// TwinCAT 3 PLC project PLC_Modbus_TCP
// ProgramVersion: 3.1.4024.0
// libraries:
//   Tc2_ModbusSrv, * (Beckhoff Automation GmbH)
//   Tc2_Standard, * (Beckhoff Automation GmbH)
//   Tc2_System, * (Beckhoff Automation GmbH)
//   Tc3_Module, * (Beckhoff Automation GmbH)
// project tree:
//   / PlcTask.TcTTO
//   POUs/ FB_Counter.TcPOU, FB_ReadCoilsExample.TcPOU, FB_WriteRegsExample.TcPOU, MAIN.TcPOU
// real-time tasks:
//   TASK PlcTask: cycle T#10ms, priority 20, ADS port 350

CONFIGURATION PLC_Modbus_TCP
    RESOURCE PLC ON TwinCAT3
        TASK PlcTask(INTERVAL := T#10ms, PRIORITY := 20);
        PROGRAM MAIN WITH PlcTask : MAIN;
    END_RESOURCE
END_CONFIGURATION

// ---- POUs/MAIN.TcPOU
PROGRAM MAIN
VAR
	fbWriteRegs : FB_WriteRegsExample;
	fbWriteRwgs_2 : FB_WriteRegsExample; 
END_VAR

fbWriteRegs();
fbWriteRwgs_2();

END_PROGRAM

// ---- POUs/FB_WriteRegsExample.TcPOU
FUNCTION_BLOCK FB_WriteRegsExample
VAR
	fbWriteRegisters : FB_MBWriteRegs;
	nWriteValueArray : ARRAY[0..9] OF INT;
	wWriteRegsValueConvertToWord : WORD;
	eWriteState : (WAIT, TRIGGER, WRITE);
	fbTriggerStart : R_TRIG;
	fbTriggerStop : R_TRIG;
	//cbLength: UINT;
	
END_VAR

fbTriggerStart();
IF fbTriggerStart.Q THEN
	IF eWriteState = WAIT THEN
		 eWriteState := TRIGGER;
	END_IF
END_IF
IF fbTriggerStop.CLK THEN
	fbWriteRegisters(bExecute := FALSE);
	eWriteState := WAIT;
END_IF
CASE eWriteState OF
	WAIT : 
	// NOTHING
	TRIGGER : 
	 //wWriteRegsValueConvertToWord := TO_WORD(nWriteValueInt);
	 (*fbWriteRegisters(
		sIPAddr:= '192.168.10.1', 
		nTCPPort:= 502, 
		nUnitID:= 16#FF, 
		nMBAddr:= 0, 
		nValue:= wWriteRegsValueConvertToWord, 
		bExecute:= TRUE, 
		tTimeout:= , 
		bBusy=> , 
		bError=> , 
		nErrId=> ); *)
	fbWriteRegisters(
		sIPAddr:= '192.168.10.1', 
		nTCPPort:= 502, 
		nUnitID:= 16#FF, 
		nQuantity:= 10, 
		nMBAddr:= 0, 
		cbLength:= SIZEOF(nWriteValueArray), 
		pSrcAddr:= ADR(nWriteValueArray), 
		bExecute:= TRUE, 
		tTimeout:= , 
		bBusy=> , 
		bError=> , 
		nErrId=> );
	eWriteState := WRITE;
	WRITE :
	fbWriteRegisters(bExecute := FALSE);
	IF NOT fbWriteRegisters.bBusy AND NOT fbWriteRegisters.bError AND NOT fbTriggerStop.CLK  THEN 
				 eWriteState := TRIGGER;
	ELSIF fbWriteRegisters.bError  THEN
 			eWriteState := WAIT;
		
	END_IF
		
END_CASE

END_FUNCTION_BLOCK

// ---- POUs/FB_Counter.TcPOU
FUNCTION_BLOCK FB_Counter
VAR
	nCounter : UDINT;
END_VAR

nCounter := nCounter + 1;

END_FUNCTION_BLOCK

// ---- POUs/FB_ReadCoilsExample.TcPOU
FUNCTION_BLOCK FB_ReadCoilsExample
VAR
	fbReadCoils : FB_MBReadCoils;
	fbReadRegisters : FB_MBReadRegs;
	nReadValue : BYTE;
	nReadRegsValue : WORD;
	eReadState : (WAIT, TRIGGER, READ);
	fbTrigger : R_TRIG;
	cbLength: UINT;
END_VAR

fbTrigger();
IF fbTrigger.Q THEN
	IF eReadState = WAIT THEN
		eReadState := TRIGGER;
	END_IF
END_IF
CASE eReadState OF
	WAIT : 
	// NOTHING
	TRIGGER : 
	(*fbReadCoils(
		sIPAddr:='192.168.10.1' , 
		nTCPPort:=502, 
		nUnitID:= 16#FF, 
		nQuantity:= 1, 
		nMBAddr:= 0, 
		cbLength:= SIZEOF(nReadValue), 
		pDestAddr:= ADR(nReadValue), 
		bExecute:= TRUE , 
		tTimeout:= , 
		bBusy=> , 
		bError=> , 
		nErrId=> , 
		cbRead=> );*)
	fbReadRegisters(
		sIPAddr:= '192.168.10.1', 
		nTCPPort:= 502, 
		nUnitID:= 16#FF, 
		nQuantity:= 1, 
		nMBAddr:= 0, 
		cbLength:= SIZEOF(nReadRegsValue), 
		pDestAddr:= ADR(nReadRegsValue), 
		bExecute:= TRUE, 
		tTimeout:= , 
		bBusy=> , 
		bError=> , 
		nErrId=> , 
		cbRead=> );
		eReadState := READ;
	READ :
	(*fbReadCoils(bExecute := FALSE);
	IF NOT fbReadCoils.bBusy OR fbReadCoils.bError THEN
		eReadState := WAIT;
	END_IF*)
	fbReadRegisters(bExecute := FALSE);
	IF NOT fbReadRegisters.bBusy AND NOT fbReadRegisters.bError THEN
		eReadState := TRIGGER;
	ELSIF fbReadRegisters.bError THEN
		eReadState := WAIT;
	END_IF
		
END_CASE

END_FUNCTION_BLOCK
